// TIA Portal V20 export
ORGANIZATION_BLOCK "CFC_Program cycle"   // OB1001, CFC, ProgramCycle
TITLE = "Main Program Sweep (Cycle)"
{ S7_Optimized_Access := 'TRUE' }
AUTHOR : CFC
FAMILY : CFCPlus
VERSION : 1.0
// stored: AutoNumber false
   VAR_INPUT
      Initial_Call : Bool;   // Initial call of this OB
      Remanence : Bool;   // =True, if remanent data are available
   END_VAR
   VAR_TEMP
      t_out : UInt;
   END_VAR
BEGIN
END_ORGANIZATION_BLOCK
